// TIA Portal V20 export
TYPE "typeEmInterlockParameters"
// stored: Access Published, Namespace Unit1
   STRUCT
      "Bool" { ExternalAccessible := 'False'; ExternalVisible := 'False'; ExternalWritable := 'False'} : Array[0..200] of Bool;
      "Dint" { ExternalAccessible := 'False'; ExternalVisible := 'False'; ExternalWritable := 'False'} : Array[0..100] of DInt;
      Lreal { ExternalAccessible := 'False'; ExternalVisible := 'False'; ExternalWritable := 'False'} : Array[0..100] of LReal;
      "Time" { ExternalAccessible := 'False'; ExternalVisible := 'False'; ExternalWritable := 'False'} : Array[0..100] of IEC_TIMER;
   END_STRUCT;
   // // "Bool"[0] : isLinked
   // // "Bool"[1] : PauseRequest
   // // "Bool"[2] : PauseDone
END_TYPE
